PROGRAM MAIN
VAR
END_VAR

END_PROGRAM

(* stored: Version 1.1.0.1
   POU MAIN: Id {60249165-1ad7-42a0-801d-d9e79a444709} *)
